(* IEC 61131-3 sources: CannyIEC/st/cannyiec/function_blocks, 3 files *)

(* ---- asymmetricdebounce-AsymmetricDebounce.st ---- *)
(* --- Interface --- *)
FUNCTION_BLOCK AsymmetricDebounce
VAR_INPUT
    IN          : BOOL;           (* raw input signal from a sensor or switch *)
    tPresetRise : TIME := T#50MS; (* preset time for rising edge debounce *)
    tPresetFall : TIME := T#50MS; (* preset time for falling edge debounce *)
END_VAR
VAR_OUTPUT
    Q : BOOL; (* debounced "input" signal *)
END_VAR
VAR
    fbDebounce : TON; (* TON instance for handling the debounce timing *)
    xWasIN     : BOOL; (* private debounced state *)
END_VAR

(* --- Implementation --- *)
(* Only accept a state change after the raw input remains stable for its
   configured debounce time. The TON runs only while the raw input differs
   from the private debounced state. *)
fbDebounce(IN := IN <> xWasIN, PT := SEL(IN, tPresetFall, tPresetRise));
IF fbDebounce.Q THEN
    xWasIN := IN;
END_IF;
Q := xWasIN;

(* ---- symmetricdebounce-SymmetricDebounce.st ---- *)
(* --- Interface --- *)
FUNCTION_BLOCK SymmetricDebounce
VAR_INPUT
    IN : BOOL;           (* raw input signal from a sensor or switch *)
    PT : TIME := T#50MS; (* preset time for rising and falling edge debounce *)
END_VAR
VAR_OUTPUT
    Q : BOOL; (* debounced "input" signal *)
END_VAR
VAR
    fbAsymmetricDebounce : AsymmetricDebounce;
END_VAR

(* --- Implementation --- *)
fbAsymmetricDebounce(IN := IN, tPresetRise := PT, tPresetFall := PT);
Q := fbAsymmetricDebounce.Q;

(* ---- trig-TRIG.st ---- *)
(* --- Interface --- *)
FUNCTION_BLOCK TRIG
VAR_INPUT
    CLK : BOOL; (* signal to monitor *)
END_VAR
VAR_OUTPUT
    Q : BOOL; (* one-cycle pulse when CLK changes *)
END_VAR
VAR
    fbRise : R_TRIG; (* rising edge trigger *)
    fbFall : F_TRIG; (* falling edge trigger *)
END_VAR

(* --- Implementation --- *)
fbRise(CLK := CLK);
fbFall(CLK := CLK);
Q := fbRise.Q OR fbFall.Q;
